KUKA KRL data list: A_ERROR.dat

&ACCESS RVO1
&REL 9
&PARAM EDITMASK = *
&PARAM TEMPLATE = C:\KRC\Roboter\Template\vorgabe
&PARAM DISKPATH = KRC:\R1\Program\HG
DEFDAT A_ERROR PUBLIC



ENDDAT
